Staubli VAL3: getSize.pgx

public program getSize(num& x_nSize[])
  local num i
  local num j
begin
  //
  // search if there are Call in the Disk
  //
  libList("",listCall)
  for i=0 to (size(listCall)-1)
    if left(listCall[i],1)!="_"
      if i==size(listCall[i])-1 and i==0
        listCall=""
      else
        delete(listCall[i])
        i=i-1
      endIf
    endIf
  endFor
  if listCall!=""
    x_nSize=size(listCall)
  else
    x_nSize=0
  endIf
end
